(* IEC 61131-3 sources: mect_apps/TP1043_RTU/ModbusRTUclient_CFG/Output, 1 file *)

(* ---- Resource1.gvl ---- *)
VAR_GLOBAL
Alarm1 AT %MD0.772:UDINT;
TPLC_OUT_1 AT %MW0.5380:INT;
TPLC_OUT_2 AT %MW0.5384:INT;
TPLC_IN_3 AT %MW0.5388:INT;
TPLC_IN_4 AT %MW0.5392:INT;
TPLC_IN_AN_1 AT %MW0.5396:INT;
TPLC_IN_AN_2 AT %MW0.5400:INT;
END_VAR
